// Mitsubishi GX Works2 project: LD_windingmachine   PLC: FX1N/FX1NC

PROGRAM MAIN
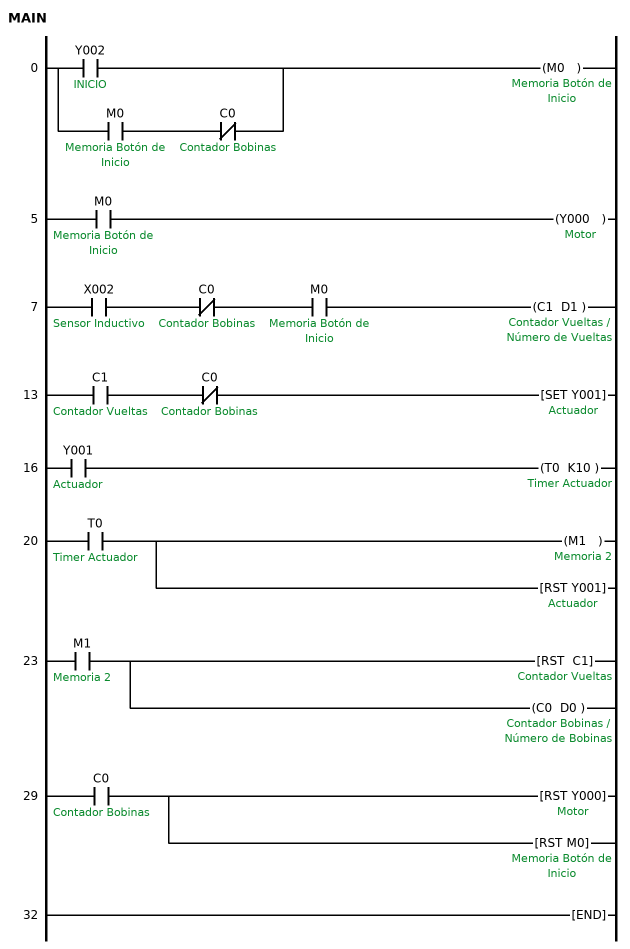
0     LD      Y002  ; INICIO
      LD      M0  ; Memoria Botón de Inicio
      ANI     C0  ; Contador Bobinas
      ORB
      OUT     M0  ; Memoria Botón de Inicio
5     LD      M0  ; Memoria Botón de Inicio
      OUT     Y000  ; Motor
7     LD      X002  ; Sensor Inductivo
      ANI     C0  ; Contador Bobinas
      AND     M0  ; Memoria Botón de Inicio
      OUT     C1 D1  ; Contador Vueltas / Número de Vueltas
13    LD      C1  ; Contador Vueltas
      ANI     C0  ; Contador Bobinas
      SET     Y001  ; Actuador
16    LD      Y001  ; Actuador
      OUT     T0 K10  ; Timer Actuador
20    LD      T0  ; Timer Actuador
      OUT     M1  ; Memoria 2
      RST     Y001  ; Actuador
23    LD      M1  ; Memoria 2
      RST     C1  ; Contador Vueltas
      OUT     C0 D0  ; Contador Bobinas / Número de Bobinas
29    LD      C0  ; Contador Bobinas
      RST     Y000  ; Motor
      RST     M0  ; Memoria Botón de Inicio
32    END
END_PROGRAM

// device comments not shown above
X000  ; Botón Inicio Principal
X001  ; Botón Inicio Bobinas
X003  ; Botón Paro
